# EPICS substitutions: modules/event/evrIoc/Db/evrPatternBP21.substitutions
#
# Pattern records
file evrPatternAll.db {
#	    Device        ,  SLC Pattern Check LNK    , EVR/Trigger
#	                                                  Links
  pattern { DEVICE        ,        LINK4               , LINK5 ,        LINK6            ,  TREF   , TS1ST, TS2ND }
	  { IOC:BP21:BP01 ,"IOC:BP21:BP01:FANOUTSLC PP",  ""   ,"IOC:BP21:BP01:FANOUT PP", 1.03E06 ,   1  ,   4   }
}
file evrEventAll.db {
  pattern { DEVICE        }
	  { IOC:BP21:BP01 }
}
